// TIA Portal V17 export
// export: Created 2025-08-05T09:36:01.4547414Z, ExportSetting WithDefaults, DisplayName Totally Integrated Automation Portal, DisplayVersion V17, DisplayName TIA Portal Openness, DisplayVersion V17, DisplayName TIA Portal Version Control Interface, DisplayVersion V17, DisplayName SINAMICS Startdrive Advanced, DisplayVersion V17, DisplayName SINAMICS Startdrive G130, G150, S120, S150, SINAMICS MV, S210, DisplayVersion V17, DisplayName SINAMICS Startdrive G110M, G120, G120C, G120D, G120P, G115D, DisplayVersion V17, DisplayName STEP 7 Professional, DisplayVersion V17, DisplayName STEP 7 Safety, DisplayVersion V17, DisplayName WinCC Advanced, DisplayVersion V17
TYPE "API_Inputs"
// stored: IsFailsafeCompliant false
   STRUCT
      Heartbeat : Bool;   // Heartbeat Input from Middleware
      Ready : Bool;   // Middleware Ready for Transations
      Job_Comp : Bool;   // Middleware Job has Been Completed
      Clear_Results : Bool;   // Clear Results Stored in PLC. Set by Middleware
      Mutex : Bool;   // Mutex Token with Middleware to Prevent Multiple Instances Running
      Rx : DInt;   // Recieved Counter
      Active_Job : DInt;   // Current Job Active in Middleware
      Fault_Code : Array[0..9] of DInt;   // Fault Code from Middleware
      Timeout : Time;   // Timeout Value for SIS Job. Value set by Middleware and is dependant upon Job Function.
      LDD : Struct   // Laser Depth Dynamics
         Ref_Plane : DInt;
         Status : Struct   // Current Status of the LDD System (Pseudo DIO)
            OK : Bool;   // LDD System is OK
            Ready_Cmd : Bool;   // LDD System is Ready to Recieve a Command
            Wait_Trigger : Bool;   // LDD System is Waiting for Trigger
            Acquiring : Bool;   // LDD System is Acquiring Data
            Remote_Control : Bool;   // LDD is in Remote Mode
            Seq_Complete : Bool;   // Overall Sequence is Complete
            Seq_Pass : Bool;   // Overall Sequence has Passed
            Seq_Fail : Bool;   // Overall Sequence has Failed
         END_STRUCT;
         DDO : Array[0.."LASERCOMM_LDD_ARRAY_SIZE"] of "LaserComm_DDO";   // Array for Storage of Measurement Data from LDD
         Results : Array[0.."LASERCOMM_LDD_ARRAY_SIZE"] of "LaserComm_LDD_Results";   // Array for Storage of LDD QA Results
      END_STRUCT;
      YLR { S7_SetPoint := 'True'} : "YLR_Inputs";   // Inputs from YLR Laser (signals handled by Middleware)
   END_STRUCT;
END_TYPE
